(* Statuses of the pumps, valves, and gauges for the for the BO4 Output tube *)
TYPE ST_TransportTubeStatuses :
STRUCT
	// Pump statuses
	bIonPumpOn : BOOL;
	
	// Valve statuses
	bGateValveOpen : BOOL;
	
	// Gauge statuses
	fPiraniGaugeVal : REAL;
	ePiraniGaugeState : E_PressureState;
	fColdCathodeVal : REAL;
	eColdCathodeState : E_PressureState;
	
END_STRUCT
END_TYPE

(* stored: Version 1.1.0.1, ProductVersion 3.1.4024.0
   DUT ST_TransportTubeStatuses: Id {aa3ada0e-610c-0be5-2cbb-33936e779cce} *)
